(* CODESYS project States.library
   Company: _
   DefaultNamespace: States
   Title: States
   Placeholder: _States
   Author: Krystian Lis et al.
   Description: State implementation.
   Version: 1.0.0

Project tree, tasks and I/O mapping:
  libraries: Broadcast, * (_); Debug, * (_); Results, * (_); Rt, * (_); Strings, * (_); Tags, * (_); Tc2_Standard, * (Beckhoff Automation GmbH); Tc2_System, * (Beckhoff Automation GmbH)
  State/
    Buffer/
      interface I_StateBuffer: Cap, Length, Pop, Push
      function block StateBuffer [ST]: Cap, Length, ToDebug, Pop, Push
    List/
      interface I_StateRepo: GetByPos, GetByTag, Cap, Length, Push
      function block StateRepo [ST]: GetByPos, GetByTag, Cap, Length, ToDebug, Push
    Machine/
      interface I_StateMachine: ChangeState, GetState
      function block StateMachine [ST]: ChangeState, Execute, GetState, Tag, ToDebug
    Manager/
      function block A_StateManager [ST]: FB_init, ToDebug
      interface I_StateManager: Get, GetOnChange, Request, Current, Pretender, Previous
      function block StateManager [ST]: Execute, FB_init, Get, GetOnChange, ToDebug, Request, Current, Pretender, Previous
    State/
      global variables CState
      interface I_State: Tag, CanActivate, CanDeactivate, OnExecute, OnExit, OnInit
      function block State [ST]: FB_init, Tag, ToDebug, CanActivate, CanDeactivate, OnExecute, OnExit, OnInit
*)

// State/State/CState
{attribute 'qualified_only'}
VAR_GLOBAL CONSTANT
	SUCCESS		: Strings.Str := 'Success';
	FAIL		: Strings.Str := 'Fail';
	SAME		: Strings.Str := 'Same';
END_VAR

// State/Buffer/I_StateBuffer
INTERFACE I_StateBuffer EXTENDS Debug.I_Debug

METHOD Cap : UDINT
VAR_INPUT
END_VAR
END_METHOD

METHOD Length : UDINT
VAR_INPUT
END_VAR
END_METHOD

METHOD Pop : Results.Result
VAR_OUTPUT
	iState			: I_State;
END_VAR
END_METHOD

METHOD Push : Results.Result
VAR_INPUT
	iState			: I_State;
END_VAR
END_METHOD

END_INTERFACE

// State/State/I_State
INTERFACE I_State EXTENDS Debug.I_Debug, Tags.I_Tagged

PROPERTY Tag : Tags.I_Tag
GET
END_GET
END_PROPERTY

METHOD CanActivate : BOOL
VAR_INPUT
END_VAR
END_METHOD

METHOD CanDeactivate : BOOL
VAR_INPUT
END_VAR
END_METHOD

METHOD OnExecute
VAR_INPUT
END_VAR
END_METHOD

METHOD OnExit
VAR_INPUT
END_VAR
END_METHOD

METHOD OnInit
VAR_INPUT
END_VAR
END_METHOD

END_INTERFACE

// State/Buffer/StateBuffer
FUNCTION_BLOCK StateBuffer
VAR_GENERIC CONSTANT
	nMax				: UDINT(0..16#FFFFFFE) := 1;
END_VAR
IMPLEMENTS I_StateBuffer
VAR
	_iState				: ARRAY[0..nMax] OF I_State;
	_nHead				: UDINT;
	_nTail				: UDINT;
	_nLen				: UDINT;

	
	_fbTagOwner			: Tags.TagOwner;
END_VAR

METHOD Cap : UDINT
VAR_INPUT
END_VAR
Cap := nMax;
END_METHOD

METHOD Length : UDINT
VAR_INPUT
END_VAR
Length := _nLen;
END_METHOD

METHOD ToDebug : Debug.I_Debug
VAR_INPUT
END_VAR
ToDebug := THIS^;
END_METHOD

METHOD Pop : Results.Result
VAR_OUTPUT
	iState			: I_State;
END_VAR
IF _nHead = _nTail THEN
    Pop := Results.None;
    RETURN;
END_IF

iState := _iState[_nHead];
_iState[_nHead] := 0;

_nHead := _nHead + 1;
_nLen := _nLen - 1;

IF _nHead > nMax THEN
    _nHead := 0;
END_IF

Pop := Results.Ok;
END_METHOD

METHOD Push : Results.Result
VAR_INPUT
	iState			: I_State;
END_VAR
VAR
	_nNextTail 		: UDINT;
END_VAR
IF iState = 0 THEN
	Push := Results.Err.Itf0;
	RETURN;
END_IF

_nNextTail := _nTail + 1;

IF _nNextTail > nMax THEN
    _nNextTail := 0;
END_IF

IF _nNextTail = _nHead THEN
    Push := Results.Err.Ovf; 
    RETURN;
END_IF

_nLen := _nLen + 1;
_iState[_nTail] := iState;
_nTail := _nNextTail;
Push := Results.Ok;
END_METHOD

END_FUNCTION_BLOCK

// State/List/I_StateRepo
INTERFACE I_StateRepo EXTENDS Debug.I_Debug

METHOD GetByPos : Results.Result
VAR_INPUT
	nPos			: UDINT;
END_VAR
VAR_OUTPUT
	iState			: I_State;
END_VAR
END_METHOD

METHOD GetByTag : Results.Result
VAR_INPUT
	iTag			: Tags.I_Tag;
END_VAR
VAR_OUTPUT
	iState			: I_State;
END_VAR
END_METHOD

METHOD Cap : UDINT
VAR_INPUT
END_VAR
END_METHOD

METHOD Length : UDINT
VAR_INPUT
END_VAR
END_METHOD

METHOD Push : Results.Result
VAR_INPUT
	iState			: I_State;
END_VAR
VAR_OUTPUT
	nPos			: UDINT;
END_VAR
END_METHOD

END_INTERFACE

// State/List/StateRepo
FUNCTION_BLOCK StateRepo
VAR_GENERIC CONSTANT
	nMax				: UDINT(0..16#FFFFFFE) := 10;
END_VAR
IMPLEMENTS I_StateRepo
VAR
	_iState				: ARRAY[0..nMax] OF I_State;
	_nLen				: UDINT;
	_fbTagOwner			: Tags.TagOwner;
END_VAR

METHOD GetByPos : Results.Result
VAR_INPUT
	nPos		: UDINT;
END_VAR
VAR_OUTPUT
	iState		: I_State;
END_VAR
IF nPos > nMax THEN
	GetByPos := Results.Err.Ovf;
	RETURN;
END_IF

iState := _iState[nPos];
IF iState <> 0 THEN
	GetByPos := Results.Ok;
END_IF
END_METHOD

METHOD GetByTag : Results.Result
VAR_INPUT
	iTag			: Tags.I_Tag;
END_VAR
VAR_OUTPUT
	iState			: I_State;
END_VAR
VAR
	_nCache			: UDINT;
	i				: UDINT;
END_VAR
IF iTag = 0 THEN
	GetByTag := Results.Err.Itf0;
	RETURN;
END_IF

IF iTag.Owner <> _fbTagOwner.Self THEN
	GetByTag := Results.Err.NoMatch;
	RETURN;
END_IF

iState := _iState[iTag.Cache];

GetByTag := Results.Ok;
END_METHOD

METHOD Cap : UDINT
VAR_INPUT
END_VAR
Cap := nMax;
END_METHOD

METHOD Length : UDINT
VAR_INPUT
END_VAR
Length := _nLen;
END_METHOD

METHOD ToDebug : Debug.I_Debug
VAR_INPUT
END_VAR
ToDebug := THIS^;
END_METHOD

METHOD Push : Results.Result
VAR_INPUT
	iState			: I_State;
END_VAR
VAR_OUTPUT
	nPos			: UDINT;
END_VAR
VAR
	_nPos			: UDINT;
END_VAR
IF iState = 0 THEN
	Push := Results.Err.Itf0;
	RETURN;
END_IF

IF nMax < _nLen THEN
	Push := Results.Err.Ovf;
	RETURN;
END_IF

IF Results.IsErr(iState.Tag.Join(_fbTagOwner, _nLen), eCarry => Push) THEN
	RETURN;
END_IF

_iState[_nLen] := iState;
_nLen := _nLen + 1;
Push := Results.Ok;
END_METHOD

END_FUNCTION_BLOCK

// State/Machine/I_StateMachine
INTERFACE I_StateMachine EXTENDS Debug.I_Debug, Tags.I_Tagged

METHOD ChangeState : Results.Result
VAR_INPUT
	iNewState	: I_State;
END_VAR
VAR_OUTPUT
	iOldState	: I_State;
END_VAR
END_METHOD

METHOD GetState : I_State
VAR_INPUT
END_VAR
END_METHOD

END_INTERFACE

// State/Machine/StateMachine
FUNCTION_BLOCK FINAL StateMachine IMPLEMENTS I_StateMachine, Rt.I_Execute
VAR
	_fbExe					: Rt.Execute(THIS^);
	_fbTag					: Tags.Tag;
	_iCurrentState			: I_State;
END_VAR

METHOD ChangeState : Results.Result
VAR_INPUT
	iNewState	: I_State;
END_VAR
VAR_OUTPUT
	iOldState	: I_State;
END_VAR
IF iNewState = 0 THEN
	_fbTag.Option := CState.FAIL;
	ChangeState := Results.Err.Itf0;
	RETURN;
END_IF

IF iNewState = _iCurrentState THEN
	_fbTag.Option := CState.SAME;
	ChangeState := Results.None;
END_IF

IF NOT iNewState.CanActivate() THEN
	_fbTag.Option := CState.FAIL;
	ChangeState := Results.None;
	RETURN;
END_IF

IF _iCurrentState <> 0 AND_THEN NOT _iCurrentState.CanDeactivate() THEN
	_fbTag.Option := CState.FAIL;
	ChangeState := Results.None;
	RETURN;
END_IF

IF _iCurrentState <> 0 THEN
	_iCurrentState.OnExit();
END_IF

iNewState.OnInit();
iOldState := _iCurrentState;
_iCurrentState := iNewState;
_fbTag.Option := CState.SUCCESS;
ChangeState := Results.Ok;
END_METHOD

METHOD Execute
IF _iCurrentState <> 0 THEN
	_iCurrentState.OnExecute();
END_IF
END_METHOD

METHOD GetState : I_State
VAR_INPUT
END_VAR
GetState := _iCurrentState;
END_METHOD

PROPERTY Tag : Tags.I_Tag
GET
END_GET
END_PROPERTY

METHOD ToDebug : Debug.I_Debug
END_METHOD

END_FUNCTION_BLOCK

// State/Manager/A_StateManager
FUNCTION_BLOCK A_StateManager IMPLEMENTS Debug.I_Debug
VAR_INPUT
END_VAR
VAR_OUTPUT
END_VAR
VAR
END_VAR

//FB_Init is always available implicitly and it is used primarily for initialization.
//The return value is not evaluated. For a specific influence, you can also declare the
//methods explicitly and provide additional code there with the standard initialization
//code. You can evaluate the return value.
METHOD FB_Init: BOOL
VAR_INPUT
    bInitRetains: BOOL; // TRUE: the retain variables are initialized (reset warm / reset cold)
    bInCopyCode: BOOL;  // TRUE: the instance will be copied to the copy code afterward (online change)   

	iStateManager		: I_StateManager;
	refStateManager		: REFERENCE TO I_StateManager;
END_VAR
IF NOT __ISVALIDREF(refStateManager) THEN
	Debug.DebugMsg(THIS^, ': Ref = 0!');
	RETURN;
END_IF

IF iStateManager = 0 THEN
	Debug.DebugMsg(THIS^, ': Itf = 0!');
	RETURN;
END_IF

IF refStateManager <> 0 THEN
	Debug.DebugMsg(THIS^, ': Ref itf should be unassigned!');
	RETURN;
END_IF

refStateManager := iStateManager;
END_METHOD

METHOD ToDebug : Debug.I_Debug
ToDebug := THIS^;
END_METHOD

END_FUNCTION_BLOCK

// State/Manager/I_StateManager
INTERFACE I_StateManager EXTENDS Debug.I_Debug

METHOD Get : Results.Result
VAR_INPUT
	nPos				: UDINT;
END_VAR
VAR_OUTPUT
	iTag				: Tags.I_Tag;
END_VAR
END_METHOD

METHOD GetOnChange : Broadcast.I_Signal
VAR_INPUT
END_VAR
END_METHOD

METHOD Request : Results.Result
VAR_INPUT
	iTag		: Tags.I_Tag;
END_VAR
END_METHOD

PROPERTY Current : Tags.I_Tag
GET
END_GET
END_PROPERTY

PROPERTY Pretender : Tags.I_Tag
GET
END_GET
END_PROPERTY

PROPERTY Previous : Tags.I_Tag
GET
END_GET
END_PROPERTY

END_INTERFACE

// State/Manager/StateManager
FUNCTION_BLOCK StateManager
VAR_GENERIC CONSTANT
	nMax				: UDINT := 10;
END_VAR
IMPLEMENTS Rt.I_Execute, I_StateManager, Debug.I_Debug

VAR
	_fbExecute			: Rt.Execute(THIS^);
	_iMachine			: I_StateMachine;
	_iRepo				: I_StateRepo;
	_iBuffer			: I_StateBuffer;
	_iBufferCached		: ARRAY[0..nMax] OF BOOL; 
	
	_iPretender			: Tags.I_Tag;
	_iCurrent			: Tags.I_Tag;
	_iPrevious 			: Tags.I_Tag;
	
	_fbOnChange			: Broadcast.Signal;
END_VAR

METHOD Execute
VAR
	_iNewState		: I_State;
	_iOldState		: I_State;
END_VAR
IF Results.IsOk(_iBuffer.Pop(iState => _iNewState)) THEN
	_iPretender := _iNewState.Tag;
	_iBufferCached[_iPretender.Cache] := FALSE;
	IF Results.IsOk(_iMachine.ChangeState(_iNewState, iOldState => _iOldState)) THEN
		_iPretender		:= 0;
		_iCurrent		:= _iNewState.Tag;
		IF _iOldState <> 0 THEN
			_iPrevious		:= _iOldState.Tag;
		END_IF
		_fbOnChange.Emit(_iMachine.Tag);
	ELSE
		_fbOnChange.Emit(_iMachine.Tag);
	END_IF
END_IF
END_METHOD

//FB_Init is always available implicitly and it is used primarily for initialization.
//The return value is not evaluated. For a specific influence, you can also declare the
//methods explicitly and provide additional code there with the standard initialization
//code. You can evaluate the return value.
METHOD FB_Init: BOOL
VAR_INPUT
    bInitRetains: BOOL; // TRUE: the retain variables are initialized (reset warm / reset cold)
    bInCopyCode: BOOL;  // TRUE: the instance will be copied to the copy code afterward (online change)
	
	iMachine		: I_StateMachine;
	iRepo			: I_StateRepo;
	iBuffer			: I_StateBuffer;
END_VAR
IF iMachine = 0 OR iBuffer = 0 OR iRepo = 0 THEN
	IF iMachine = 0 THEN
		Debug.DebugMsg(THIS^, Tc2_Standard.CONCAT(__POUNAME(), ': Initialized with null iStateMachine: I_StateMachine!'));	
	END_IF
	IF iBuffer = 0 THEN
		Debug.DebugMsg(THIS^, Tc2_Standard.CONCAT(__POUNAME(), ': Initialized with null iBuffer: I_StateList!'));	
	END_IF
	IF iRepo = 0 THEN
		Debug.DebugMsg(THIS^, Tc2_Standard.CONCAT(__POUNAME(), ': Initialized with null iRepo: I_StateList!'));
	END_IF
	RETURN;
END_IF

_iMachine := iMachine;
_iBuffer := iBuffer;
_iRepo := iRepo;
END_METHOD

METHOD Get : Results.Result
VAR_INPUT
	nPos				: UDINT;
END_VAR
VAR_OUTPUT
	iTag				: Tags.I_Tag;
END_VAR
VAR
	_iState				: I_State;
END_VAR
IF Results.IsOk(_iRepo.GetByPos(nPos, iState => _iState), eCarry => Get) THEN
	iTag := _iState.Tag;
END_IF
END_METHOD

METHOD GetOnChange : Broadcast.I_Signal
VAR_INPUT
END_VAR
GetOnChange := _fbOnChange;
END_METHOD

METHOD ToDebug : Debug.I_Debug
ToDebug := THIS^;
END_METHOD

METHOD Request : Results.Result
VAR_INPUT
	iTag		: Tags.I_Tag;
END_VAR
VAR
	_iState		: I_State;
END_VAR
IF NOT Results.IsOk(_iRepo.GetByTag(iTag, iState => _iState), eCarry => Request) THEN
	RETURN;
END_IF

IF _iBufferCached[iTag.Cache] THEN
	Request := Results.Ok;
	RETURN;
END_IF

_iBufferCached[iTag.Cache] := TRUE;

Request := _iBuffer.Push(_iState);
END_METHOD

PROPERTY Current : Tags.I_Tag
GET
Current := _iCurrent;
END_GET
END_PROPERTY

PROPERTY Pretender : Tags.I_Tag
GET
Pretender := _iPretender;
END_GET
END_PROPERTY

PROPERTY Previous : Tags.I_Tag
GET
Previous := _iPrevious;
END_GET
END_PROPERTY

END_FUNCTION_BLOCK

// State/State/State
FUNCTION_BLOCK ABSTRACT State IMPLEMENTS I_State
VAR
	_fbTag						: Tags.Tag;
END_VAR

//FB_Init is always available implicitly and it is used primarily for initialization.
//The return value is not evaluated. For a specific influence, you can also declare the
//methods explicitly and provide additional code there with the standard initialization
//code. You can evaluate the return value.
METHOD FB_Init: BOOL
VAR_INPUT
    bInitRetains: BOOL; // TRUE: the retain variables are initialized (reset warm / reset cold)
    bInCopyCode: BOOL;  // TRUE: the instance will be copied to the copy code afterward (online change)
	
	iStateList					: I_StateRepo;
END_VAR
IF iStateList = 0 THEN
	Debug.DebugMsg(THIS^, Tc2_Standard.CONCAT(__POUNAME(), ': Itf = 0!'));
	RETURN;
END_IF

CASE iStateList.Push(THIS^) OF
	Results.Ok:
		// No Error
	Results.None:
		Debug.DebugMsg(iStateList.ToDebug(), Tc2_Standard.CONCAT(__POUNAME(), ': Tried to insert a double!'));
		Debug.DebugMsg(THIS^, 'Im a double!');
	Results.Err.Ovf:
		Debug.DebugMsg(iStateList.ToDebug(), Tc2_Standard.CONCAT(__POUNAME(), ': Overflow!'));
		Debug.DebugMsg(THIS^, 'Cause of overflow!');
	Results.Err.NoMatch:
		Debug.DebugMsg(iStateList.ToDebug(), Tc2_Standard.CONCAT(__POUNAME(), ': No Match!'));
		Debug.DebugMsg(THIS^, 'This already have an owner!');
	ELSE
		Debug.DebugMsg(iStateList.ToDebug(), Tc2_Standard.CONCAT(__POUNAME(), ': Unknown Error!'));
		Debug.DebugMsg(THIS^, 'Cause!');		
END_CASE
END_METHOD

PROPERTY Tag : Tags.I_Tag
GET
Tag := _fbTag;
END_GET
END_PROPERTY

METHOD ToDebug : Debug.I_Debug
ToDebug := THIS^;
END_METHOD

METHOD CanActivate : BOOL
VAR_INPUT
END_VAR
CanActivate := TRUE;
END_METHOD

METHOD CanDeactivate : BOOL
VAR_INPUT
END_VAR
CanDeactivate := TRUE;
END_METHOD

METHOD OnExecute
VAR_INPUT
END_VAR
END_METHOD

METHOD OnExit
VAR_INPUT
END_VAR
END_METHOD

METHOD OnInit
VAR_INPUT
END_VAR
END_METHOD

END_FUNCTION_BLOCK
